PROGRAM UpdateSys
VAR
	SysUpdate_R1			:FB_UpdateSys;
	SysUpdate_R2			:FB_UpdateSys;
	SysUpdate_R3			:FB_UpdateSys;
	SysUpdate_R4			:FB_UpdateSys;
	SysUpdate_R5			:FB_UpdateSys;
	SysUpdate_R6			:FB_UpdateSys;
	SysUpdate_R7			:FB_UpdateSys;
END_VAR

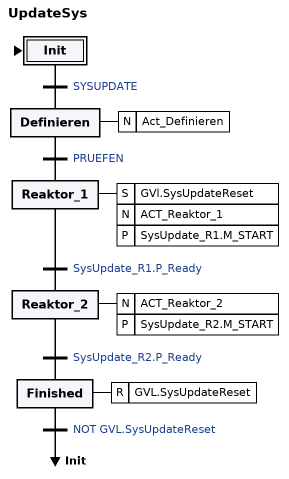
INITIAL_STEP Init:
END_STEP
TRANSITION FROM Init TO Definieren
    := SYSUPDATE;
END_TRANSITION
STEP Definieren:
    Act_Definieren(N);
END_STEP
TRANSITION FROM Definieren TO Reaktor_1
    := PRUEFEN;
END_TRANSITION
STEP Reaktor_1:
    GVl.SysUpdateReset(S);
    ACT_Reaktor_1(N);
    SysUpdate_R1.M_START(P);
END_STEP
TRANSITION FROM Reaktor_1 TO Reaktor_2
    := SysUpdate_R1.P_Ready;
END_TRANSITION
STEP Reaktor_2:
    ACT_Reaktor_2(N);
    SysUpdate_R2.M_START(P);
END_STEP
TRANSITION FROM Reaktor_2 TO Finished
    := SysUpdate_R2.P_Ready;
END_TRANSITION
STEP Finished:
    GVL.SysUpdateReset(R);
END_STEP
TRANSITION FROM Finished TO Init
    := NOT GVL.SysUpdateReset;
END_TRANSITION

ACTION ACT_Definieren:
IF GVL.SysUpdate_1 THEN
	IF GVL.R1_SW.ReactReady <> GVL.SysStatusWord.R1_Ready THEN
		GVL.SysStatusWord.R1_Ready := GVL.R1_SW.ReactReady;
	END_IF
	
	IF GVL.R1_SW.ReactActiv <> GVL.SysStatusWord.R1_Activ THEN
		GVL.SysStatusWord.R1_Activ := GVL.R1_SW.ReactActiv;
	END_IF
END_IF

IF GVL.SysUpdate_2 THEN
	IF GVL.R2_SW.ReactReady <> GVL.SysStatusWord.R2_Ready THEN
		GVL.SysStatusWord.R2_Ready := GVL.R2_SW.ReactReady;
	END_IF
	
	IF GVL.R2_SW.ReactActiv <> GVL.SysStatusWord.R2_Activ THEN
		GVL.SysStatusWord.R2_Activ := GVL.R2_SW.ReactActiv;
	END_IF
END_IF

IF GVL.SysUpdate_3 THEN
	IF GVL.R3_SW.ReactReady <> GVL.SysStatusWord.R3_Ready THEN
		GVL.SysStatusWord.R3_Ready := GVL.R3_SW.ReactReady;
	END_IF
	
	IF GVL.R3_SW.ReactActiv <> GVL.SysStatusWord.R3_Activ THEN
		GVL.SysStatusWord.R3_Activ := GVL.R3_SW.ReactActiv;
	END_IF
END_IF

IF GVL.SysUpdate_4 THEN
	IF GVL.R4_SW.ReactReady <> GVL.SysStatusWord.R4_Ready THEN
		GVL.SysStatusWord.R4_Ready := GVL.R4_SW.ReactReady;
	END_IF
	
	IF GVL.R4_SW.ReactActiv <> GVL.SysStatusWord.R4_Activ THEN
		GVL.SysStatusWord.R4_Activ := GVL.R4_SW.ReactActiv;
	END_IF
END_IF

IF GVL.SysUpdate_5 THEN
	IF GVL.R5_SW.ReactReady <> GVL.SysStatusWord.R5_Ready THEN
		GVL.SysStatusWord.R5_Ready := GVL.R5_SW.ReactReady;
	END_IF
	
	IF GVL.R5_SW.ReactActiv <> GVL.SysStatusWord.R5_Activ THEN
		GVL.SysStatusWord.R5_Activ := GVL.R5_SW.ReactActiv;
	END_IF
END_IF

IF GVL.SysUpdate_6 THEN
	IF GVL.R6_SW.ReactReady <> GVL.SysStatusWord.R6_Ready THEN
		GVL.SysStatusWord.R6_Ready := GVL.R6_SW.ReactReady;
	END_IF
	
	IF GVL.R6_SW.ReactActiv <> GVL.SysStatusWord.R6_Activ THEN
		GVL.SysStatusWord.R6_Activ := GVL.R6_SW.ReactActiv;
	END_IF
END_IF

IF GVL.SysUpdate_7 THEN
	IF GVL.R7_SW.ReactReady <> GVL.SysStatusWord.R7_Ready THEN
		GVL.SysStatusWord.R7_Ready := GVL.R7_SW.ReactReady;
	END_IF
	
	IF GVL.R7_SW.ReactActiv <> GVL.SysStatusWord.R7_Activ THEN
		GVL.SysStatusWord.R7_Activ := GVL.R7_SW.ReactActiv;
	END_IF
END_IF
END_ACTION

ACTION ACT_Reaktor_1:
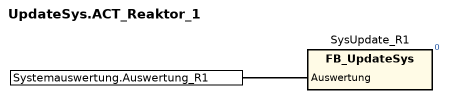
SysUpdate_R1(Auswertung := Systemauswertung.Auswertung_R1); // FB_UpdateSys
END_ACTION

ACTION ACT_Reaktor_2:
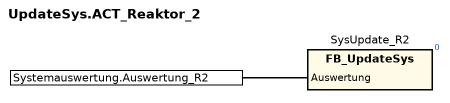
SysUpdate_R2(Auswertung := Systemauswertung.Auswertung_R2); // FB_UpdateSys
END_ACTION

TRANSITION PRUEFEN:
IF GVL.SysUpdate_1 THEN
	IF GVL.R1_SW.ReactReady = GVL.SysStatusWord.R1_Ready AND GVL.R1_SW.ReactActiv = GVL.SysStatusWord.R1_Activ THEN
		PRUEFEN := TRUE;
	ELSE
		PRUEFEN := FALSE;
	END_IF
END_IF

IF GVL.SysUpdate_2 THEN
	IF GVL.R2_SW.ReactReady = GVL.SysStatusWord.R2_Ready AND GVL.R2_SW.ReactActiv = GVL.SysStatusWord.R2_Activ THEN
		PRUEFEN := TRUE;
	ELSE
		PRUEFEN := FALSE;
	END_IF
END_IF

IF GVL.SysUpdate_3 THEN
	IF GVL.R3_SW.ReactReady = GVL.SysStatusWord.R3_Ready AND GVL.R3_SW.ReactActiv = GVL.SysStatusWord.R3_Activ THEN
		PRUEFEN := TRUE;
	ELSE
		PRUEFEN := FALSE;
	END_IF
END_IF

IF GVL.SysUpdate_4 THEN
	IF GVL.R4_SW.ReactReady = GVL.SysStatusWord.R4_Ready AND GVL.R4_SW.ReactActiv = GVL.SysStatusWord.R4_Activ THEN
		PRUEFEN := TRUE;
	ELSE
		PRUEFEN := FALSE;
	END_IF
END_IF

IF GVL.SysUpdate_5 THEN
	IF GVL.R5_SW.ReactReady = GVL.SysStatusWord.R5_Ready AND GVL.R5_SW.ReactActiv = GVL.SysStatusWord.R5_Activ THEN
		PRUEFEN := TRUE;
	ELSE
		PRUEFEN := FALSE;
	END_IF
END_IF

IF GVL.SysUpdate_6 THEN
	IF GVL.R6_SW.ReactReady = GVL.SysStatusWord.R6_Ready AND GVL.R6_SW.ReactActiv = GVL.SysStatusWord.R6_Activ THEN
		PRUEFEN := TRUE;
	ELSE
		PRUEFEN := FALSE;
	END_IF
END_IF

IF GVL.SysUpdate_7 THEN
	IF GVL.R7_SW.ReactReady = GVL.SysStatusWord.R7_Ready AND GVL.R7_SW.ReactActiv = GVL.SysStatusWord.R7_Activ THEN
		PRUEFEN := TRUE;
	ELSE
		PRUEFEN := FALSE;
	END_IF
END_IF
END_TRANSITION

TRANSITION SYSUPDATE:
IF GVL.SysUpdate_1 OR
	GVL.SysUpdate_2 OR
	GVL.SysUpdate_3 OR
	GVL.SysUpdate_4 OR
	GVL.SysUpdate_5 OR
	GVL.SysUpdate_6 OR
	GVL.SysUpdate_7 THEN
	
	SYSUPDATE := TRUE;
ELSE 
	SYSUPDATE := FALSE;
END_IF
END_TRANSITION

END_PROGRAM

(* stored: Version 1.1.0.1, ProductVersion 3.1.4024.12
   POU UpdateSys: Id {274d45d6-f99e-48d7-a8bf-62705c3dba75}, SpecialFunc None
   Folder 01_Aktionen: Id {34fb21c4-2429-47c7-bd45-a946093ef632}
   Folder 02_Transitionen: Id {c9094467-c1d7-4cf2-9493-8d42202b9700}
   Action ACT_Definieren: Id {e6c2213a-af8d-4420-91e9-52d730b27633}
   Action ACT_Reaktor_1: Id {eb2bb236-841f-414f-ac59-87afb8702e25}
   Action ACT_Reaktor_2: Id {3d258a9a-c4ff-49a2-81b0-e41bae662cd0}
   Transition PRUEFEN: Id {4292ae78-7b13-4f7f-9166-589699e46f33}
   Transition SYSUPDATE: Id {7fba60dd-dc8a-43eb-a884-b0b41cd01dc8} *)
